FUNCTION_BLOCK ErrorTrack IMPLEMENTS iTrack
VAR_INPUT
END_VAR
VAR_OUTPUT
END_VAR
VAR
END_VAR

PROPERTY CurrentMoverCount : DINT
GET


ADSLOGSTR( ADSLOG_MSGTYPE_ERROR, 'The Track.GetCurrentMoverCount property as accessed on an error track.', '');
END_GET
END_PROPERTY

PROPERTY CurrentMoverList : iMoverList
GET


ADSLOGSTR( ADSLOG_MSGTYPE_ERROR, 'The Track.GetCurrentMoverList property as accessed on an error track.', '');
END_GET
END_PROPERTY

PROPERTY Id : INT
GET


ADSLOGSTR( ADSLOG_MSGTYPE_ERROR, 'The Track.Id get property is unavailable while the mover is activating a new track.', '');
END_GET
SET


ADSLOGSTR( ADSLOG_MSGTYPE_ERROR, 'The Track.Id set property is unavailable while the mover is activating a new track.', '');
END_SET
END_PROPERTY

PROPERTY OTCID : OTCID
GET


ADSLOGSTR( ADSLOG_MSGTYPE_ERROR, 'The Track.OTCID get property is unavailable while the mover is activating a new track.', '');
END_GET
SET


ADSLOGSTR( ADSLOG_MSGTYPE_ERROR, 'The Track.OTCID set property is unavailable while the mover is activating a new track.', '');
END_SET
END_PROPERTY

METHOD RegisterMover : BOOL
VAR_INPUT
    NewMover : REFERENCE TO Mover;
END_VAR
VAR
	i : ULINT;
END_VAR


ADSLOGSTR( ADSLOG_MSGTYPE_ERROR, 'The Track.RegisterMover function was called on an error track.', '');
END_METHOD

METHOD UnregisterAll : BOOL
VAR_INPUT
END_VAR


ADSLOGSTR( ADSLOG_MSGTYPE_ERROR, 'The Track.UnregisterAll function was called on an error track.', '');
END_METHOD

METHOD UnregisterMover : BOOL
VAR_INPUT
    RemovingMover : REFERENCE TO Mover;
END_VAR
VAR
	i : ULINT;
END_VAR


ADSLOGSTR( ADSLOG_MSGTYPE_ERROR, 'The Track.UnregisterMover function was called on an error track.', '');
END_METHOD

END_FUNCTION_BLOCK

(* stored: Version 1.1.0.1, ProductVersion 3.1.4024.12
   POU ErrorTrack: Id {b7d2262d-2290-026e-04de-e41a4d953470}, SpecialFunc None
   Folder Methods: Id {eeff0d3e-8d73-0d64-379f-cf0d456afc19}
   Folder Properties: Id {13bdc662-fc7c-04cc-21a6-3ca65662fecd}
   Property CurrentMoverCount: Id {33bc7799-5276-0c26-1ca1-9d07d364e1a1}
   Get Get: Id {ed94d4d3-8277-0713-23f5-a3ff80dd5525}
   Property CurrentMoverList: Id {b190691f-b4b8-0ba1-0821-763dc5d8bf10}
   Get Get: Id {f7bc1d95-fb88-0b8f-0c46-ca2451a3ca1b}
   Property Id: Id {3f245ec6-2d35-0e07-007d-ee805d2b4910}
   Get Get: Id {8bf80f8b-c4c5-033d-3938-7faf2a4b2089}
   Set Set: Id {08d650b4-e18a-001a-1529-9066b9b74657}
   Property OTCID: Id {ddf37bf7-b48a-0af3-260c-7b9e319896e8}
   Get Get: Id {c7411707-c9da-00e0-065a-2c6b4c6ba42b}
   Set Set: Id {de34ce6f-78eb-003b-21a4-99278d48bb7c}
   Method RegisterMover: Id {4c665ebf-fb7e-0a21-2133-e9b3f174b407}
   Method UnregisterAll: Id {b731f48b-54fa-0a81-0269-2584465b6ef9}
   Method UnregisterMover: Id {c64abf39-b0cc-091a-0a6a-5a9c47d60b9d} *)
